FUNCTION_BLOCK ReqPanelLift (* Composite Function Block Type *)
  (* Standard: 61499-2 *)
  (* Version 0.0, 6/3/2016, Andrei, nxtControl GmbH, template *)
  PACKAGE Main;
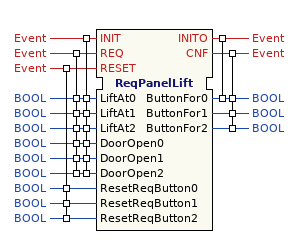
  EVENT_INPUT
    INIT WITH LiftAt0, LiftAt1, LiftAt2, DoorOpen0, DoorOpen1, DoorOpen2; (* Initialization Request *)
    REQ WITH LiftAt0, LiftAt1, LiftAt2, DoorOpen0, DoorOpen1, DoorOpen2; (* Normal Execution Request *)
    RESET WITH ResetReqButton0, ResetReqButton1, ResetReqButton2;
  END_EVENT
  EVENT_OUTPUT
    INITO WITH ButtonFor0; (* Initialization Confirm *)
    CNF WITH ButtonFor0, ButtonFor1, ButtonFor2; (* Execution Confirmation *)
  END_EVENT
  VAR_INPUT
    LiftAt0 : BOOL; (* Input event qualifier *)
    LiftAt1 : BOOL;
    LiftAt2 : BOOL;
    DoorOpen0 : BOOL;
    DoorOpen1 : BOOL;
    DoorOpen2 : BOOL;
    ResetReqButton0 : BOOL;
    ResetReqButton1 : BOOL;
    ResetReqButton2 : BOOL;
  END_VAR
  VAR_OUTPUT
    ButtonFor0 : BOOL; (* Output event qualifier *)
    ButtonFor1 : BOOL;
    ButtonFor2 : BOOL;
  END_VAR
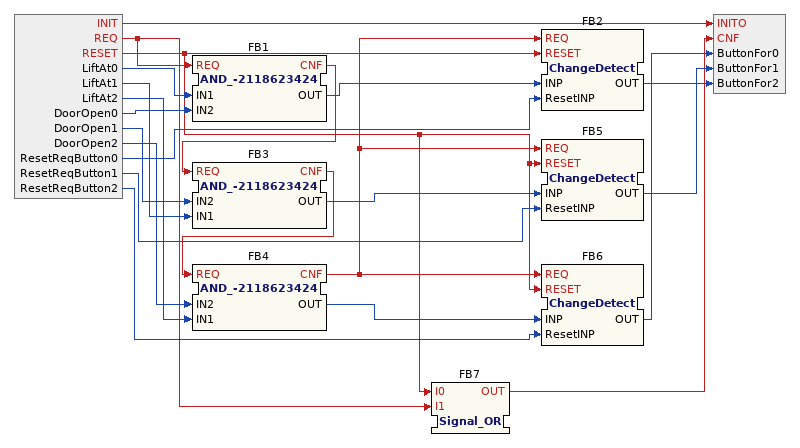
  FBS
    FB1 : AND_-2118623424; {SET_ATTRIBUTE(Configuration.GenericFBType.InterfaceParams, Runtime.Standard#CNT:=2;OUT:BOOL)}
    FB3 : AND_-2118623424; {SET_ATTRIBUTE(Configuration.GenericFBType.InterfaceParams, Runtime.Standard#CNT:=2;OUT:BOOL)}
    FB4 : AND_-2118623424; {SET_ATTRIBUTE(Configuration.GenericFBType.InterfaceParams, Runtime.Standard#CNT:=2;OUT:BOOL)}
    FB7 : Signal_OR;
    FB2 : ChangeDetect;
    FB5 : ChangeDetect;
    FB6 : ChangeDetect;
  END_FBS
  EVENT_CONNECTIONS
    REQ TO FB1.REQ;
    FB1.CNF TO FB3.REQ;
    FB3.CNF TO FB4.REQ;
    FB4.CNF TO FB6.REQ;
    FB4.CNF TO FB5.REQ;
    FB4.CNF TO FB2.REQ;
    RESET TO FB2.RESET;
    RESET TO FB5.RESET;
    RESET TO FB6.RESET;
    RESET TO FB7.I0;
    FB7.OUT TO CNF;
    INIT TO INITO;
    REQ TO FB7.I1;
  END_CONNECTIONS
  DATA_CONNECTIONS
    LiftAt0 TO FB1.IN1;
    DoorOpen0 TO FB1.IN2;
    DoorOpen1 TO FB3.IN2;
    LiftAt1 TO FB3.IN1;
    DoorOpen2 TO FB4.IN2;
    LiftAt2 TO FB4.IN1;
    FB1.OUT TO FB2.INP;
    FB3.OUT TO FB5.INP;
    FB4.OUT TO FB6.INP;
    ResetReqButton0 TO FB2.ResetINP;
    ResetReqButton1 TO FB5.ResetINP;
    ResetReqButton2 TO FB6.ResetINP;
    FB2.OUT TO ButtonFor0;
    FB5.OUT TO ButtonFor1;
    FB6.OUT TO ButtonFor2;
  END_CONNECTIONS
END_FUNCTION_BLOCK
